(*********************************** G.D S.p.A. - Technical Department ***********************************
============= PROGRAM INFO ============
FOLDER:             TBD
MACHINES INVOLVED:  TBD 

============= DESCRIPTION =============

============= REVISIONS ===============
Date		Version	 	Author      	Description             
----------	-------		------------  	--------------------------------------------
2019/04/24 	0000.00	 	M.Grasso		Creation of the PRG

**********************************************************************************************************)
(*$R 
	process_ref:= prc; 
$*)
PROGRAM csp_case_main_safety_drives_SD10300
VAR
	prc:					process;
	prc_path:				STRING;	

	sig:												safety_integrated_group;
	chA_smes_sis:										safety_integrated_series;
	chB_smes_sis:										safety_integrated_series;
	safety_integrated_series_close_dvr_chA: 			BOOL;
	safety_integrated_series_close_dvr_chB: 			BOOL;

	shutdown_chA AT %Q* 								:BOOL := TRUE;
	shutdown_chB AT %Q* 								:BOOL := TRUE;
END_VAR

_read_var_input();

_objects_manager();

IF NOT objects_running()
THEN
	RETURN;	
END_IF

_read_process_image();

_mode_manager();

//safety_integrated_series_close(chA_smes_sis);
//safety_integrated_series_close(chB_smes_sis);

IF  safety_integrated_series_get_mode (chA_smes_sis) = MODE_ABSENT
	OR
	safety_integrated_series_get_mode(chA_smes_sis) = MODE_INACTIVE
	THEN
		shutdown_chA := TRUE;
	ELSE
		shutdown_chA := FALSE;
END_IF

IF  safety_integrated_series_get_mode (chB_smes_sis) = MODE_ABSENT
	OR
	safety_integrated_series_get_mode(chB_smes_sis) = MODE_INACTIVE
	THEN
		shutdown_chB := TRUE;
	ELSE
		shutdown_chB := FALSE;
END_IF

CASE process_get_mode(prc) OF
	MODE_ABSENT,
	MODE_INACTIVE:
		RETURN;
	MODE_TEST:
		;
END_CASE

_set_runtime_properties();

(********************************* BODY *********************************)
IF NOT safety_integrated_group_is_running(sig)
		THEN
			safety_integrated_group_run(sig);
END_IF
safety_integrated_series_close(chA_smes_sis);
safety_integrated_series_close(chB_smes_sis);
safety_integrated_series_close_dvr_chA := safety_integrated_series_is_safely_closed(chA_smes_sis);
safety_integrated_series_close_dvr_chB := safety_integrated_series_is_safely_closed(chB_smes_sis);
(************************************************************************)

_handle_messages();

_write_output();

ACTION _handle_messages:
;
END_ACTION

ACTION _handle_process_test:
;
END_ACTION

ACTION _mode_manager:
IF process_mode_req_is_pending(prc)
THEN
    process_apply_mode_req_first_step(prc);
    CASE process_get_mode(prc) OF
        MODE_TO_ABSENT:
			;
        MODE_TO_INACTIVE:
			;
        MODE_TO_TEST:
			;
        MODE_TO_OPERATIONAL:
			;
    END_CASE
    process_apply_mode_req_second_step(prc);
END_IF
END_ACTION

ACTION _objects_manager:
IF objects_initialization()
THEN
	sub_process_init(
		object_name					:= 'csp_case_main_safety_drives.prc', 
		process						:= csp_case_main_safety_drives.prc, 
		CONVERSION_this				:= prc);
		
	prc_path 						:= process_get_path(prc);

	safety_integrated_group_init(
        object_name				:=	CONCAT(prc_path, '_sig'), 
		controller				:=	csp_case_main_safety_interface.SPLC5000_sic,
        process					:=	prc,
        CONVERSION_this			:=	sig);

	(* Channel A SMES series *)
	safety_integrated_series_init(
		object_name				:=	CONCAT(prc_path, '_chA_smes_sis'), 
		_type					:=	SAFETY_INTEGRATED_SERIES_TYPE_NO_RESET,
		discrepancy_active		:=	TRUE,
		forced_open_active		:=	TRUE,
		process					:=	prc,
		CONVERSION_this			:=	chA_smes_sis);

	safety_integrated_series_add_safety_integrated_group(
		group					:=	sig,
		CONVERSION_this			:=	chA_smes_sis);

	safety_integrated_series_add_safety_integrated_series(
		series_active			:=	TRUE,
		series_polarity_direct	:=	TRUE,
		contact					:=	csp_case_main_safety_drives_commonConfiguration.rack_smes_sis, (*Marco : To be checked*)
		CONVERSION_this			:=	chA_smes_sis);
		
	(* Channel B SMES series *)
	safety_integrated_series_init(
		object_name				:=	CONCAT(prc_path, '_chB_smes_sis'), 
		_type					:=	SAFETY_INTEGRATED_SERIES_TYPE_NO_RESET,
		discrepancy_active		:=	TRUE,
		forced_open_active		:=	TRUE,
		process					:=	prc,
		CONVERSION_this			:=	chB_smes_sis);

	safety_integrated_series_add_safety_integrated_group(
		group					:=	sig,
		CONVERSION_this			:=	chB_smes_sis);
		
	safety_integrated_series_add_safety_integrated_series(
		series_active			:=	TRUE,
		series_polarity_direct	:=	TRUE,
		contact					:=	csp_case_main_safety_drives_commonConfiguration.rack_smes_sis, (*Marco : To be checked*)
		CONVERSION_this			:=	chB_smes_sis);
		
END_IF

IF objects_running()
THEN
	process_cycle(prc);
  	safety_integrated_group_cycle(sig);
	safety_integrated_series_cycle(chA_smes_sis);
	safety_integrated_series_cycle(chB_smes_sis);
END_IF
END_ACTION

ACTION _read_process_image:
;
END_ACTION

ACTION _read_var_input:
;
END_ACTION

ACTION _set_runtime_properties:
;
END_ACTION

ACTION _write_output:
;
END_ACTION

END_PROGRAM

(* stored: Version 1.1.0.1, ProductVersion 3.1.4024.3
   POU csp_case_main_safety_drives_SD10300: Id {a57ea087-5c8b-4a0f-9113-28ed495495e5}, SpecialFunc None
   Action _handle_messages: Id {623ec3ba-d57e-4af0-825e-a3d1f3a5d045}
   Action _handle_process_test: Id {d260a386-0173-42a2-bab9-24c77971e464}
   Action _mode_manager: Id {7854e606-ebb7-4c29-8b6f-5d1f2cfb0f23}
   Action _objects_manager: Id {eeb1fce6-9211-4a88-a538-b7ae1281e715}
   Action _read_process_image: Id {0e8df8ef-a630-4815-915d-231f0ac9ff56}
   Action _read_var_input: Id {fa0146c3-59a0-432b-aa7e-49c0439c49a4}
   Action _set_runtime_properties: Id {70b59318-1827-428f-885c-f188a42aacf8}
   Action _write_output: Id {7a9959a2-326a-451f-8561-44d7a78efb0d} *)
